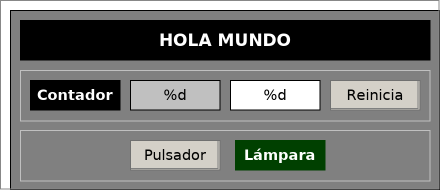
VISUALIZATION V_Hola_Mundo  // 440x190
    Rectangle (10,10 430x180)
    Rectangle (20,70 410x51)
    Rectangle (20,130 410x51)
    Rectangle (20,20 410x40), "HOLA MUNDO"
    Rectangle (30,80 90x30), "Contador"
    Rectangle (230,80 90x30), "%d", text variable: MAIN.ContadorCiclos
        OnMouseClick: write the text variable via Default
    Rectangle (130,80 90x30), "%d", text variable: MAIN.ContadorCiclos
    Button (330,80 90x30), "Reinicia"
        OnMouseClick: execute { MAIN.ContadorCiclos := 0; }
    Button (130,140 90x30), "Pulsador"
        tap MAIN.i_Pulsador
    Rectangle (235,140 90x30), "Lámpara", colour toggle: MAIN.o_Lampara
END_VISUALIZATION

(* stored: Version 1.1.0.1, ProductVersion 3.1.4024.16
   Visu V_Hola_Mundo: Id {29eb6263-18b7-411e-9454-972d0b476675} *)
